// TIA Portal V17 export
// export: Created 2024-08-07T21:44:12.4030065Z, ExportSetting WithDefaults, DisplayName Totally Integrated Automation Portal, DisplayVersion V17 Update 7, DisplayName TIA Portal Openness, DisplayVersion V17 Update 7, DisplayName TIA Portal Version Control Interface, DisplayVersion V17, DisplayName SINAMICS Startdrive Advanced, DisplayVersion V17 SP2, DisplayName SINAMICS Startdrive G110M, G120, G120C, G120D, G120P, G115D, DisplayVersion V17 SP2, DisplayName SINAMICS Startdrive G130, G150, S120, S150, SINAMICS MV, S210, DisplayVersion V17 SP2, DisplayName STEP 7 Professional, DisplayVersion V17 Update 7, DisplayName STEP 7 Safety, DisplayVersion V17 Update 6, DisplayName WinCC Advanced / Unified PC, DisplayVersion V17 Update 7
VAR_GLOBAL   // PLC tag table "plc"
   iAirPressure AT %I0.1 : Bool;
   iEmergencyStopHydraulics1 AT %I1.0 : Bool;
   iEmergencyStopHydraulics2 AT %I1.1 : Bool;
   iBtnOpenServiceDoors1 AT %I1.2 : Bool;
   iBtnResetServiceDoors1 AT %I1.3 : Bool;
   iBtnOpenServiceDoors2 AT %I1.4 : Bool;
   iBtnResetServiceDoors2 AT %I1.5 : Bool;
   qServiceDoorUnlock1 AT %Q1.0 : Bool;
   qServiceDoorUnlock2 AT %Q1.1 : Bool;
   qLighthouseRed AT %Q1.3 : Bool;
   qLighthouseOrange AT %Q1.4 : Bool;
   qLighthouseGreen AT %Q1.6 : Bool;
   qLighthouseWhite AT %Q1.7 : Bool;
   qLEDDoors1Open AT %Q3.0 : Bool;
   qLEDDoors2Open AT %Q3.1 : Bool;
   qLEDDoors1EMG AT %Q3.3 : Bool;
   qLEDDoors2EMG AT %Q3.4 : Bool;
   iAntennaStartCycle AT %I0.0 : Bool;
   qMS6reset AT %Q3.6 : Bool;
   qResetServiceDoors AT %Q0.1 : Bool;
   qSafetyScannerReset AT %Q0.2 : Bool;
   qLEDsafetyScannerReset AT %Q1.2 : Bool;
   iSafetyScannerResetNotRequired AT %I2.7 : Bool;
   iServiceDoorClosed1 AT %I1.6 : Bool;
   iServiceDoorClosed2 AT %I1.7 : Bool;
   qAudioSignal AT %Q0.0 : Bool;
   qLighthouseBlue AT %Q1.5 : Bool;
   iEmergencyStopConveyor AT %I2.3 : Bool;
END_VAR
